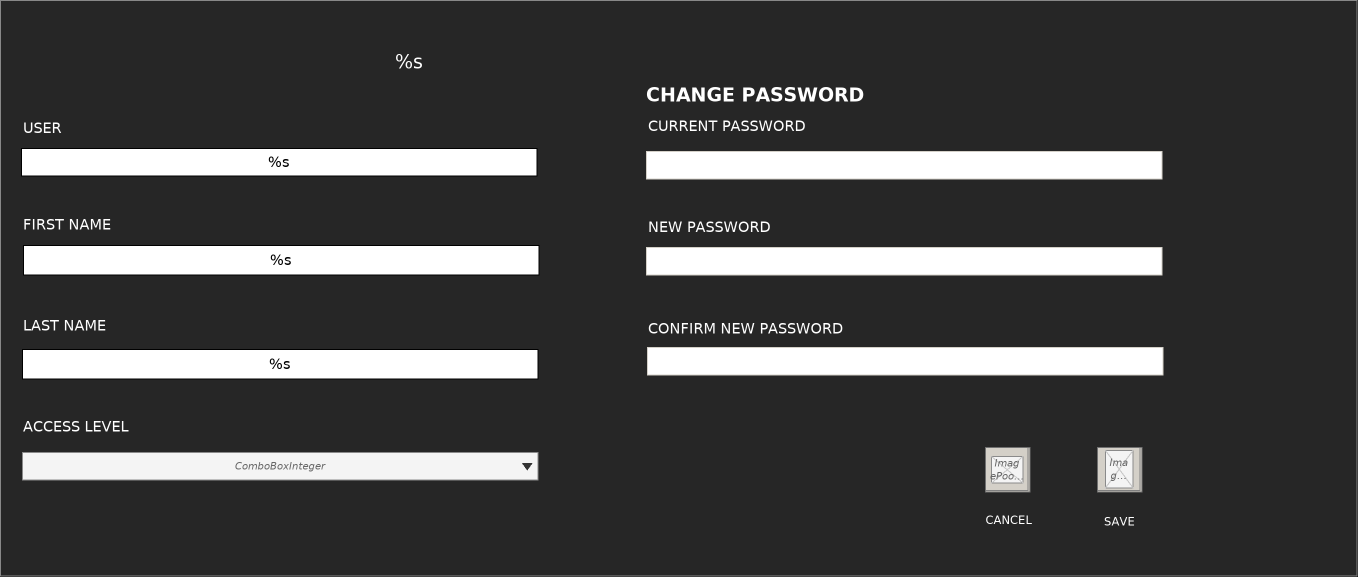
VISUALIZATION Edit_User  // 1358x577
    Rectangle (0,0 1358x577)
    Label (20,400 216x53), "ACCESS LEVEL"
    Label (20,299 216x53), "LAST NAME"
    Label (20,97 123x62), "USER"
    Label (20,198 216x53), "FIRST NAME"
    Label (643,76 417x38), "CHANGE PASSWORD"
    Label (645,196 195x62), "NEW PASSWORD"
    Label (645,302 230x53), "CONFIRM NEW PASSWORD"
    Textfield (647,347 516x28), text variable: sUM_ConfirmPassword
        OnMouseDown: write the text variable via Default, password
    Textfield (646,247 516x28), text variable: sUM_NewPassword
        OnMouseDown: write the text variable via Default, password
    Group (1077,447 85x99)
        toggle bUM_ConfirmPB
        OnMouseDown: toggle bUserNameEditPageOn
        Button (20,0 45x45)
        Label (0,50 85x49), "SAVE"
        Image (28,3 28x38), image: ImagePool.Save Button
    Group (954,447 110x102)
        toggle bUM_ReturnPB
        OnMouseDown: toggle bUserNameEditPageOn
        Button (31,0 45x45)
        Label (0,44 110x58), "CANCEL"
        Image (37,9 32x27), image: ImagePool.Delete User
    Label (645,95 195x62), "CURRENT PASSWORD"
    Textfield (646,151 516x28), text variable: sUM_CurrentPassword
        OnMouseDown: write the text variable via Default, password
    Rectangle (21,148 516x28), "%s", text variable: sUM_NewUserFirstName
        OnMouseDown: write the text variable via Default
    Rectangle (23,245 516x30), "%s", text variable: sUM_NewUserFirstName
        OnMouseDown: write the text variable via Default
    Rectangle (22,349 516x30), "%s", text variable: sUM_NewUserLastName
        OnMouseDown: write the text variable via Default
    Textfield (25,47 768x30), "%s", text variable: sMessage
    ComboBoxInteger (22,452 516x28), variable: sUM_NewUserGroupId, text list: 'TextList_AccessLevel'
END_VISUALIZATION

(* stored: Version 1.1.0.1, ProductVersion 3.1.4024.12
   Visu Edit_User: Id {402e2c1f-8f17-494f-a109-6b3055929707} *)
